// TIA Portal V20 export
FUNCTION "DTLToString" : String   // FC20220, LAD
{ S7_Optimized_Access := 'TRUE' }
// stored: AutoNumber false, SetENOAutomatically false
   VAR_INPUT
      inDTL : DTL;   // Date as DTL tag
   END_VAR
   VAR_TEMP
      format : Bool;   // 1 = traditional, 0 = international
      separatorDate : Char;   // Separator between date components
      tempString : String;   // -
      tempSepTime : Char;   // -
      tempSepTimeNano : Char;   // -
      tempPosYear : USInt;   // -
      tempPosMonth : USInt;   // -
      tempPosDay : USInt;   // -
      tempPosHour : USInt;   // -
      tempPosMinute : USInt;   // -
      tempPosSecond : USInt;   // -
      tempPosNanosecond : USInt;   // -
      tempPosSepYearMonth : USInt;   // -
      tempPosSepMonthDay : USInt;   // -
      tempPosSepHourMinute : USInt;   // -
      tempPosSepMinuteSecond : USInt;   // -
      tempPosSepSecondNanosecond : USInt;   // -
      tempCount : Int;   // -
   END_VAR
BEGIN

REGION Network 1 (SCL): Initialization
   #tempString := '';
   #tempSepTime := ':';
   #tempSepTimeNano := '.';
   #format := 1;
END_REGION

REGION Network 2 (SCL): Set format parameters for output string
   IF  #format
   THEN                                          // International ISO 8601
       #tempPosYear := 1;                          // DTL  | Y| Y| Y| Y| -| M| M| -| D| D|  | H| H| :| M| M| :| S| S| .|NS|NS|NS|NS|NS|NS|NS|NS|NS
       #tempPosMonth := 6;                         // -----|--|--|--|--|--|--|--|--|--|--|--|--|--|--|--|--|--|--|--|--|--|--|--|--|--|--|--|--|--
       #tempPosDay := 9;                           // Pos  | 1| 2| 3| 4| 5| 6| 7| 8| 9|10|11|12|13|14|15|16|17|18|19|20|21|22|23|24|25|26|27|28|29
       #tempPosHour := 12;
       #tempPosMinute := 15;
       #tempPosSecond := 18;
       #tempPosNanosecond := 21;
       #tempPosSepYearMonth := 5;
       #tempPosSepMonthDay := 8;
       #tempPosSepHourMinute := 14;
       #tempPosSepMinuteSecond := 17;
       #tempPosSepSecondNanosecond := 20;
   ELSE                                          // Traditional (EU)
       #tempPosYear := 7;                          // DTL  | D| D| -| M| M| -| Y| Y| Y| Y|  | H| H| :| M| M| :| S| S| .|NS|NS|NS|NS|NS|NS|NS|NS|NS
       #tempPosMonth := 4;                         // -----|--|--|--|--|--|--|--|--|--|--|--|--|--|--|--|--|--|--|--|--|--|--|--|--|--|--|--|--|--
       #tempPosDay := 1;                           // Pos  | 1| 2| 3| 4| 5| 6| 7| 8| 9|10|11|12|13|14|15|16|17|18|19|20|21|22|23|24|25|26|27|28|29
       #tempPosHour := 12;
       #tempPosMinute := 15;
       #tempPosSecond := 18;
       #tempPosNanosecond := 21;
       #tempPosSepYearMonth := 6;
       #tempPosSepMonthDay := 3;
       #tempPosSepHourMinute := 14;
       #tempPosSepMinuteSecond := 17;
       #tempPosSepSecondNanosecond := 20;
   END_IF;
END_REGION

REGION Network 3 (SCL): Convert "Value" into "String" and place at the right position
   //==> DTL YEAR --> String --> #tempPosYear
   VAL_STRG(FORMAT := W#16#0000,
            IN := #inDTL.YEAR,
            P := #tempPosYear,
            PREC := 0,
            SIZE := 4,
            OUT => #tempString);    
   //==> DTL MONTH --> String --> #tempPosMonth
   VAL_STRG(FORMAT := W#16#0000,
            IN := #inDTL.MONTH,
            P := #tempPosMonth,
            PREC := 0,
            SIZE := 2,
            OUT => #tempString);     
   //==> DTL DAY --> String --> #tempPosDay
   VAL_STRG(FORMAT := W#16#0000,
            IN := #inDTL.DAY,
            P := #tempPosDay,
            PREC := 0,
            SIZE := 2,
            OUT => #tempString);    
   //==> DTL HOUR --> String --> #tempPosHour
   VAL_STRG(FORMAT := W#16#0000,
            IN := #inDTL.HOUR,
            P := #tempPosHour,
            PREC := 0,
            SIZE := 2,
            OUT => #tempString);     
   //==> DTL MINUTE --> String --> #tempPosMinute
   VAL_STRG(FORMAT := W#16#0000,
            IN := #inDTL.MINUTE,
            P := #tempPosMinute,
            PREC := 0,
            SIZE := 2,
            OUT => #tempString);     
   //==> DTL SECOND --> String --> #tempPosSecond
   VAL_STRG(FORMAT := W#16#0000,
            IN := #inDTL.SECOND,
            P := #tempPosSecond,
            PREC := 0,
            SIZE := 2,
            OUT => #tempString);     
   //==> // DTL NANOSECOND --> String --> #tempPosNanosecond
   VAL_STRG(FORMAT := W#16#0000,
            IN := #inDTL.NANOSECOND,
            P := #tempPosNanosecond,
            PREC := 0,
            SIZE := 9,
            OUT => #tempString);
END_REGION

REGION Network 4 (SCL): Place separators at the right position in the string
   #tempString[#tempPosSepYearMonth] := #separatorDate;
   #tempString[#tempPosSepMonthDay] := #separatorDate;
   #tempString[#tempPosSepHourMinute] := #tempSepTime;
   #tempString[#tempPosSepMinuteSecond] := #tempSepTime;
   #tempString[#tempPosSepSecondNanosecond] := #tempSepTimeNano;
END_REGION

REGION Network 5 (SCL): Correcting the string, due to the conversion of a leading "0" value into a "blank".-
   //==> Replacing of "blank" by "0"
   IF (#tempString[#tempPosMonth] = ' ')
   THEN
       #tempString[#tempPosMonth] := '0';
   END_IF;

   IF (#tempString[#tempPosDay] = ' ')
   THEN
       #tempString[#tempPosDay] := '0';
   END_IF;

   IF (#tempString[#tempPosHour] = ' ')
   THEN
       #tempString[#tempPosHour] := '0';
   END_IF;

   IF (#tempString[#tempPosMinute] = ' ')
   THEN
       #tempString[#tempPosMinute] := '0';
   END_IF;

   IF (#tempString[#tempPosSecond] = ' ')
   THEN
       #tempString[#tempPosSecond] := '0';
   END_IF;
END_REGION

REGION Network 6 (SCL): Temp count
   FOR #tempCount := 0 TO 5 BY 1
   DO
       IF (#tempString[#tempPosNanosecond + #tempCount] = ' ')
       THEN
           #tempString[#tempPosNanosecond + #tempCount] := '0';
       ELSE
           EXIT;
       END_IF;
   END_FOR;
END_REGION

REGION Network 7 (SCL): DTL to string
   #DTLToString := #tempString;
END_REGION
END_FUNCTION
